// SIMATIC S7-200 SMART project (STEP 7-Micro/WIN SMART), CPU ST40

SYMBOL_TABLE System Symbols
Always_On        SM0.0    // Always ON
First_Scan_On    SM0.1    // ON for the first scan cycle only
HSC0_Ctrl        SMB37    // Configure and control HSC0
HSC0_CV          SMD38    // HSC0 new current value
HSC0_PV          SMD42    // HSC0 new preset value
END_SYMBOL_TABLE

ORGANIZATION_BLOCK MAIN:OB1
TITLE=Program Comments
BEGIN
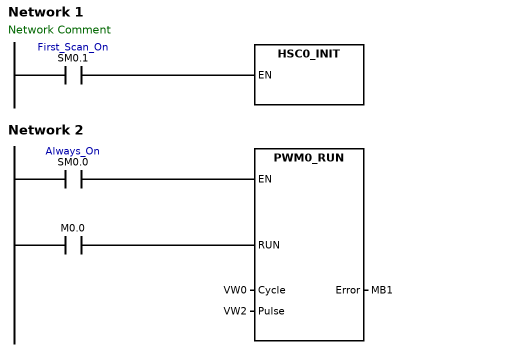
Network 1
// Network Comment
LD     First_Scan_On:SM0.1
CALL   HSC0_INIT:SBR1
Network 2
LD     Always_On:SM0.0
=      L60.0
LD     M0.0
=      L63.7
LD     L60.0
CALL   PWM0_RUN:SBR2, L63.7, VW0, VW2, MB1
END_ORGANIZATION_BLOCK

SUBROUTINE_BLOCK HSC0_INIT:SBR1
TITLE=
BEGIN
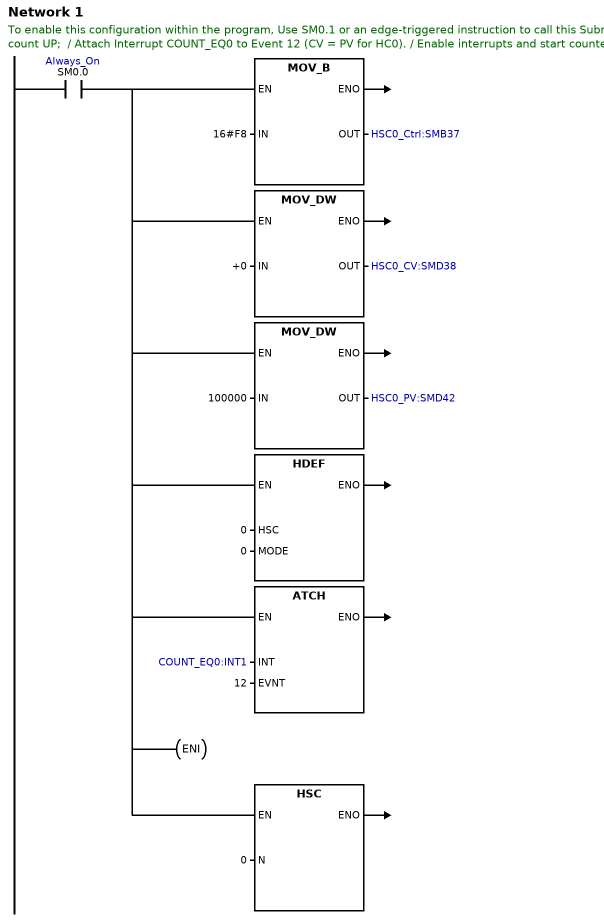
Network 1
// To enable this configuration within the program, Use SM0.1 or an edge-triggered instruction to call this Subroutine once from the MAIN program block.  
// Configure HC0 for Mode 0; CV = 0; PV = 10; count UP; 
// Attach Interrupt COUNT_EQ0 to Event 12 (CV = PV for HC0).
// Enable interrupts and start counter.
// 
//Set control bits: count UP; enabled; 
//Load CV
//Load PV
//Interrupt COUNT_EQ0: CV = PV for HC0
LD     Always_On:SM0.0
MOVB   16#F8, HSC0_Ctrl:SMB37
MOVD   +0, HSC0_CV:SMD38
MOVD   100000, HSC0_PV:SMD42
HDEF   0, 0
ATCH   COUNT_EQ0:INT1, 12
ENI
HSC    0
END_SUBROUTINE_BLOCK

// SBR2: protected block, not included

INTERRUPT_BLOCK COUNT_EQ0:INT1
TITLE=
BEGIN
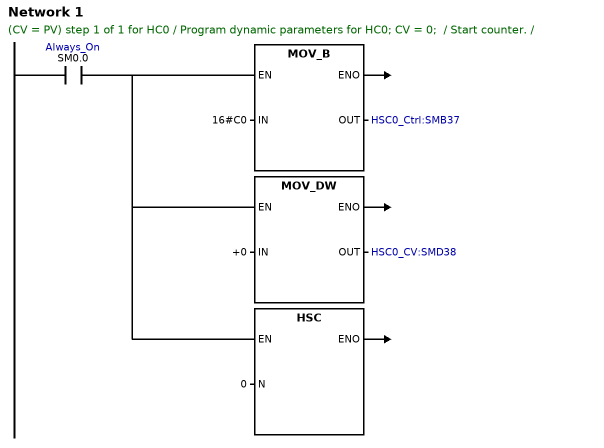
Network 1
// (CV = PV) step 1 of 1 for HC0
// Program dynamic parameters for HC0; CV = 0; 
// Start counter.
// 
//Set control bits: write current; 
//CV = 0; 
LD     Always_On:SM0.0
MOVB   16#C0, HSC0_Ctrl:SMB37
MOVD   +0, HSC0_CV:SMD38
HSC    0
END_INTERRUPT_BLOCK

DATA_BLOCK_TAB Page_1
BEGIN
//DATA PAGE COMMENTS
//Press F1 for help and example data page
VW0      1000
VW2      500
END_DATA_BLOCK_TAB
